KUKA KRL data list: masref_user.dat

&ACCESS RVO1
&REL 26
&COMMENT Mastering Reference User Program
&PARAM DISKPATH = KRC:\R1\Program
DEFDAT  masref_user
;FOLD EXTERNAL DECLARATIONS;%{PE}%MKUKATPBASIS,%CEXT,%VCOMMON,%P
;FOLD GRIPPERTECH EXT
EXT  H50 (INT  :IN,INT  :IN,INT  :IN,GRP_TYP  :IN )
;ENDFOLD (GRIPPERTECH EXT)
;FOLD SPOTTECH EXT
EXT  USERSPOT (S_COMMAND  :IN,SPOT_TYPE  :IN )
;ENDFOLD (SPOTTECH EXT)
;FOLD BASISTECH EXT;%{PE}%MKUKATPBASIS,%CEXT,%VEXT,%P
EXT  BAS (BAS_COMMAND  :IN,REAL  :IN )
;ENDFOLD (BASISTECH EXT)
;FOLD USER EXT;%{E}%MKUKATPUSER,%CEXT,%VEXT,%P
;Make here your modifications

;ENDFOLD (USER EXT)
;ENDFOLD (EXTERNAL DECLERATIONS)
DECL BASIS_SUGG_T LAST_BASIS={POINT1[] "P0                      ",POINT2[] "P0                      ",CP_PARAMS[] "CPDAT0                  ",PTP_PARAMS[] "PDAT0                   ",CONT[] "                        ",CP_VEL[] "1                       ",PTP_VEL[] "100                     ",SYNC_PARAMS[] "SYNCDAT                 ",SPL_NAME[] "S0                      ",A_PARAMS[] "ADAT0                   "}
DECL E6POS XREF_POS={X 723.753601,Y -907.651855,Z 694.200867,A -17.4627037,B 47.9882927,C 88.1239395,S 6,T 58,E1 0.0,E2 0.0,E3 0.0,E4 0.0,E5 0.0,E6 0.0}
DECL FDAT FRef_Pos={TOOL_NO 0,BASE_NO 0,IPO_FRAME #BASE,POINT2[] " ",TQ_STATE FALSE}
DECL LDAT LCPDAT1={VEL 2.00000,ACC 100.000,APO_DIST 100.000,APO_FAC 50.0000,AXIS_VEL 100.000,AXIS_ACC 100.000,ORI_TYP #VAR,CIRC_TYP #BASE,JERK_FAC 50.0000,GEAR_JERK 50.0000,EXAX_IGN 0}
DECL E6POS XAPPROACH={X 447.568420,Y -847.605042,Z 648.780212,A -21.4534302,B 49.0170898,C 91.7607880,S 6,T 58,E1 0.0,E2 0.0,E3 0.0,E4 0.0,E5 0.0,E6 0.0}
DECL FDAT FApproach={TOOL_NO 0,BASE_NO 0,IPO_FRAME #BASE,POINT2[] " ",TQ_STATE FALSE}
DECL PDAT PPDAT1={VEL 100.000,ACC 100.000,APO_DIST 100.000,GEAR_JERK 50.0000,EXAX_IGN 0}
DECL E6POS XP1={X 589.251953,Y -473.064941,Z 1226.70593,A -8.84024048,B 15.5102825,C 42.1471214,S 6,T 58,E1 0.0,E2 0.0,E3 0.0,E4 0.0,E5 0.0,E6 0.0}
DECL FDAT FP1={TOOL_NO 0,BASE_NO 0,IPO_FRAME #BASE,POINT2[] " ",TQ_STATE FALSE}
DECL PDAT PPDAT2={VEL 100.000,ACC 100.000,APO_DIST 100.000,GEAR_JERK 50.0000,EXAX_IGN 0}
DECL PDAT PPDAT3={VEL 100.000,ACC 100.000,APO_DIST 100.000,GEAR_JERK 50.0000,EXAX_IGN 0}
DECL LDAT LCPDAT2={VEL 2.00000,ACC 100.000,APO_DIST 100.000,APO_FAC 50.0000,AXIS_VEL 100.000,AXIS_ACC 100.000,ORI_TYP #VAR,CIRC_TYP #BASE,JERK_FAC 50.0000,GEAR_JERK 50.0000,EXAX_IGN 0}
DECL E6POS XP2={X 323.017700,Y -675.749268,Z 1173.09143,A -33.2838287,B 5.02120686,C 67.8807144,S 6,T 58,E1 0.0,E2 0.0,E3 0.0,E4 0.0,E5 0.0,E6 0.0}
DECL FDAT FP2={TOOL_NO 0,BASE_NO 0,IPO_FRAME #BASE,POINT2[] " ",TQ_STATE FALSE}
DECL PDAT PPDAT4={VEL 100.000,ACC 100.000,APO_DIST 100.000,GEAR_JERK 50.0000,EXAX_IGN 0}
DECL LDAT LCPDAT3={VEL 2.00000,ACC 100.000,APO_DIST 100.000,APO_FAC 50.0000,AXIS_VEL 100.000,AXIS_ACC 100.000,ORI_TYP #VAR,CIRC_TYP #BASE,JERK_FAC 50.0000,GEAR_JERK 50.0000,EXAX_IGN 0}
DECL PDAT PPDAT0={VEL 100.000,ACC 100.000,APO_DIST 100.000,GEAR_JERK 50.0000,EXAX_IGN 0}
DECL E6POS XP0={X 827.683899,Y 5.09658813,Z 1137.84778,A 166.068283,B 45.0030479,C 89.9634781,S 6,T 50,E1 0.0,E2 0.0,E3 0.0,E4 0.0,E5 0.0,E6 0.0}
DECL FDAT FP0={TOOL_NO 0,BASE_NO 0,IPO_FRAME #BASE,POINT2[] " ",TQ_STATE FALSE}
DECL PDAT PPDAT5={VEL 100.000,ACC 100.000,APO_DIST 100.000,GEAR_JERK 50.0000,EXAX_IGN 0}
DECL E6POS XP3={X 827.683899,Y 5.09658813,Z 747.698120,A 166.068283,B 45.0030479,C 89.9634781,S 6,T 50,E1 0.0,E2 0.0,E3 0.0,E4 0.0,E5 0.0,E6 0.0}
DECL FDAT FP3={TOOL_NO 0,BASE_NO 0,IPO_FRAME #BASE,POINT2[] " ",TQ_STATE FALSE}
DECL PDAT PPDAT6={VEL 100.000,ACC 100.000,APO_DIST 100.000,GEAR_JERK 50.0000,EXAX_IGN 0}
DECL LDAT LCPDAT4={VEL 2.00000,ACC 100.000,APO_DIST 100.000,APO_FAC 50.0000,AXIS_VEL 100.000,AXIS_ACC 100.000,ORI_TYP #VAR,CIRC_TYP #BASE,JERK_FAC 50.0000,GEAR_JERK 50.0000,EXAX_IGN 0}
DECL PDAT PPDAT7={VEL 100.000,ACC 100.000,APO_DIST 100.000,GEAR_JERK 50.0000,EXAX_IGN 0}
DECL E6POS XP4={X 827.683899,Y 5.09658813,Z 747.698120,A 166.068283,B 45.0030479,C 89.9634781,S 6,T 50,E1 0.0,E2 0.0,E3 0.0,E4 0.0,E5 0.0,E6 0.0}
DECL FDAT FP4={TOOL_NO 0,BASE_NO 0,IPO_FRAME #BASE,POINT2[] " ",TQ_STATE FALSE}
DECL PDAT PPDAT8={VEL 100.000,ACC 100.000,APO_DIST 100.000,GEAR_JERK 50.0000,EXAX_IGN 0}
DECL E6POS XP5={X 827.683899,Y 5.09658813,Z 1137.84778,A 166.068283,B 45.0030479,C 89.9634781,S 6,T 50,E1 0.0,E2 0.0,E3 0.0,E4 0.0,E5 0.0,E6 0.0}
DECL FDAT FP5={TOOL_NO 0,BASE_NO 0,IPO_FRAME #BASE,POINT2[] " ",TQ_STATE FALSE}
DECL LDAT LCPDAT5={VEL 2.00000,ACC 100.000,APO_DIST 100.000,APO_FAC 50.0000,AXIS_VEL 100.000,AXIS_ACC 100.000,ORI_TYP #VAR,CIRC_TYP #BASE,JERK_FAC 50.0000,GEAR_JERK 50.0000,EXAX_IGN 0}
DECL LDAT LCPDAT6={VEL 2.00000,ACC 100.000,APO_DIST 100.000,APO_FAC 50.0000,AXIS_VEL 100.000,AXIS_ACC 100.000,ORI_TYP #VAR,CIRC_TYP #BASE,JERK_FAC 50.0000,GEAR_JERK 50.0000,EXAX_IGN 0}
DECL LDAT LCPDAT7={VEL 2.00000,ACC 100.000,APO_DIST 100.000,APO_FAC 50.0000,AXIS_VEL 100.000,AXIS_ACC 100.000,ORI_TYP #VAR,CIRC_TYP #BASE,JERK_FAC 50.0000,GEAR_JERK 50.0000,EXAX_IGN 0}
ENDDAT
